{attribute 'qualified_only'}
{attribute 'strict'}
TYPE ePowerstate :
(
	Charging := -1,
	None := 0,
	Discharging := 1		
)INT;
END_TYPE

(* stored: Version 1.1.0.1, ProductVersion 3.1.4026.18
   DUT ePowerstate: Id {fc55dab1-ca74-4cc0-b8b1-ee44b890f1f8} *)
